// TwinCAT 3 PLC project XboxControllerUtilities
// Title: XboxControllerUtilities
// Company: Beckhoff Community
// Author: John Helfrich
// ProjectVersion: 1.5
// Description: A library to communicate with the ADS Gamepad Service
// ProgramVersion: 3.1.4026.24
// libraries:
//   Tc2_MC2, * (Beckhoff Automation GmbH)
//   Tc2_Standard, * (Beckhoff Automation GmbH)
//   Tc2_System, * (Beckhoff Automation GmbH)
//   Tc3_Module, * (Beckhoff Automation GmbH)
//   Tc3_XPlanarStandard, * (Beckhoff Automation GmbH)
// project tree:
//   DUTs/NC/ ST_Xbox_Button_NC_Options.TcDUT (not stored), ST_Xbox_NC_Halt_Dynamics.TcDUT (not stored), ST_Xbox_1D_Joystick_NC_Options.TcDUT (not stored), ST_Xbox_2D_Joystick_NC_Options.TcDUT (not stored), ST_Xbox_Trigger_NC_Options.TcDUT (not stored)
//   DUTs/Xbox/ E_Xbox_Controller_Battery_Levels.TcDUT (not stored), E_Xbox_Controller_Battery_Types.TcDUT (not stored), ST_Xbox_Class_Command_Status.TcDUT (not stored), ST_Xbox_Controller_ADS_Inputs.TcDUT (not stored), ST_Xbox_Controller_Buttons.TcDUT (not stored), ST_Xbox_Controller_DPad.TcDUT (not stored), ST_Xbox_Controller_Joystick.TcDUT (not stored), ST_Xbox_Controller_Rumble.TcDUT (not stored), ST_Xbox_Controller_Status.TcDUT (not stored)
//   DUTs/Xbox/LowerLevel/ ST_Xbox_Controller_Buttons_Bits.TcDUT (not stored), ST_Xbox_Controller_State_Bits.TcDUT (not stored)
//   DUTs/XPlanar/ E_Xbox_XPlanar_JogMode.TcDUT (not stored), ST_Xbox_2D_Joystick_XPlanar_Options.TcDUT (not stored)
//   FBs/Xbox/ FB_Xbox_Controller.TcPOU (not stored)
//   FBs/NC/Buttons/ FB_Xbox_Single_Button_NC.TcPOU (not stored), FB_Xbox_Dual_Button_NC.TcPOU (not stored)
//   FBs/NC/Joysticks/ FB_Xbox_2D_Joystick_NC.TcPOU (not stored), FB_Xbox_1D_Joystick_NC.TcPOU (not stored)
//   FBs/NC/Triggers/ FB_Xbox_Dual_Trigger_NC.TcPOU (not stored), FB_Xbox_Single_Trigger_NC.TcPOU (not stored)
//   FBs/XPlanar/ FB_Xbox_2D_Joystick_XPlanar.TcPOU (not stored)
//   Project Information/ F_GetCompany.TcPOU (not stored), F_GetTitle.TcPOU (not stored), F_GetVersion.TcPOU (not stored)
//   Version/ Global_Version.TcGVL

// ---- Version/Global_Version.TcGVL
{attribute 'TcGenerated'}
{attribute 'no-analysis'}
{attribute 'linkalways'}
// This function has been automatically generated from the project information.
VAR_GLOBAL CONSTANT
	{attribute 'const_non_replaced'}
	stLibVersion_XboxControllerUtilities : ST_LibVersion := (iMajor := 1, iMinor := 5, iBuild := 0, iRevision := 0, nFlags := 0, sVersion := '1.5');
END_VAR
